# B&R Automation Studio project AxisControl
Automation Studio 4.12.5.95 SP; Templates  para control de eje Maestro y eje esclavo; technology packages: Acp10Arnc0 5.24.1

## Configuration Config1

CPU X20CP1586, AutomationRuntime B4.93, Build 4.1.2, Vc V4.73.1

### Task classes (Cpu.sw)
```
NcDataObjects: acp10etxen <- AxisObjects.acp10etxen.dob, VAxInit <- AxisObjects.Virtual.VAxInit.dob, AcpParTab <- AxisObjects.Real.AcpParTab.dob, AxInit <- AxisObjects.Real.AxInit.dob
Libraries: Acp10man, Acp10par, NcGlobal, Acp10sim, Acp10_MC, sys_lib, brsystem, runtime, MpAxis, MpBase, MpCom
```

### Hardware
```
8BVIxxxxxxDx.xxx-x : 8BVIxxxxxxDx.xxx-x v2.3.0.1  [PLK1 -> X20CP1586.IF3 (NodeNumber=1) [Cable Type=PowerlinkCable, Length=10, Version=1.0.0.3]]
  MotionTP = Acp10Arnc0
  Simulate = standard
X20CP1586 : X20CP1586 v1.10.0.0
  Connector IF2:
    ActivateDevice = 1
  ConfigurationID = AxisControl_Config1
  Simulation = 1
  TimerDeviceType = EPLX2X
  TimerDevice = X20CP1586.IF3
  TaskClassIdleTime = 2000
  FileDevice1
  FileDeviceName1 = USER
  FileDevicePath1 = USER_PATH
```

### Acp10cfg.ncc - X20CP1586/Motion/Acp10cfg.ncc
```
NcConfiguration (Version=5.24.1, NcSwId=Acp10)
  ACP10CF1_typ:
    cnt_nettrc_rec_drive = 1500
    bufsize_trace_upload = 1200
    tc_nc_man_task = Cyclic #1
    glob_pv_as_ncobject = Yes
    ncsys_dl_broadcast = Yes
    ncsys_dl_acp_reset = Yes
    safemc_log_err_to_ax = Yes
    network_init:
      ncsw_init_execute = Yes
      automatic_execute = No
      node_nr_warning = Yes
      net_err_before_ncact = Yes
    nettrc:
      enter_parsecrec = Yes
      enter_ncaction = Yes
      save_ring_startidx = Yes
    cam_prof_download:
      cam_dat_dl_parallel = No
      tc_cam_dl_parallel = Task class for NC Manager task
    plk_if[0]:
      if_name = IF3
      tc_CycDat_PLCopen = Task class for NC Manager task
      mc_broadcast_extdat = No
```

### Acp10map.ncm - X20CP1586/Motion/Acp10map.ncm
```
NcMapping (NcSwId=Acp10, DisabledNodesAreHidden=False)
  NcObject gAxis01 (ModuleId=8BVIxxxxxxDx.xxx-x, Type=ncAXIS, Channel=1, AcoposSimulation=Off, InitParameter=AxInit, AcoposParameter=AcpParTab, Disabled=FALSE, ModuleDisabled=FALSE)
  NcObject gAxis02 (ModuleId=8BVIxxxxxxDx.xxx-x, Type=ncAXIS, Channel=2, AcoposSimulation=Off, InitParameter=AxInit, AcoposParameter=AcpParTab, Disabled=FALSE, ModuleDisabled=FALSE)
  NcObject gVMaster (ModuleId=8BVIxxxxxxDx.xxx-x, Type=ncV_AXIS, Channel=1, InitParameter=VAxInit, Disabled=FALSE, ModuleDisabled=FALSE)
  NcObject gVStep (ModuleId=8BVIxxxxxxDx.xxx-x, Type=ncV_AXIS, Channel=2, InitParameter=VAxInit, Disabled=FALSE, ModuleDisabled=FALSE)
```

### Config.mpaxisbasic - X20CP1586/Motion/Config.mpaxisbasic
```
Element gVMasterLink (Type=mpaxisbasic)
  AxisConfiguration = AxisWithConfiguration
    Drive:
      Controller:
        LoopFilters:
          [0]
          [1]
          [2]
Element gVStepLink (Type=mpaxisbasic)
  AxisConfiguration = AxisWithConfiguration
    Drive:
      Controller:
        LoopFilters:
          [0]
          [1]
          [2]
Element gRealAxisLink_1 (Type=mpaxisbasic)
  AxisConfiguration = AxisWithConfiguration
    Drive:
      Controller:
        LoopFilters:
          [0]
          [1]
          [2]
Element gRealAxisLink_2 (Type=mpaxisbasic)
  AxisConfiguration = AxisWithConfiguration
    Drive:
      Controller:
        LoopFilters:
          [0]
          [1]
          [2]
```

## Logical view

Binary libraries used (declarations not repeated): operator, runtime, astime, AsIecCon, Acp10man, Acp10par, NcGlobal, Acp10sim, Acp10_MC, sys_lib, brsystem, MpAxis, MpBase, MpCom, standard

### Global.typ - Global data types
```iecst
TYPE
	Axis_type : 	STRUCT
		Enable : BOOL; (*Habilita Control Global del eje*)
		Cmd : AxisComand_type;
		Sts : AxisStatus_type;
		Par : AxisParameters_type;
	END_STRUCT;
	AxisComand_type : 	STRUCT
		Enable : BOOL;
		Reset : BOOL;
		ConfigReq : BOOL;
	END_STRUCT;
	AxisStatus_type : 	STRUCT
		ConfigDone : BOOL;
		Error : BOOL;
	END_STRUCT;
	AxisParameters_type : 	STRUCT
		New_Member : USINT;
	END_STRUCT;
END_TYPE
```

### Global.var - Global variables
```iecst
(*Declariacion Ejes *)
VAR
	gAxis01 : ACP10AXIS_typ;
	gAxis02 : ACP10AXIS_typ;
	gVMaster : ACP10VAXIS_typ;
	gVStep : ACP10VAXIS_typ;
END_VAR
(*UDT Control dej Eje*)
VAR
	gAxis : ARRAY[0..MAX_AXIS] OF Axis_type;
END_VAR
```

### Constant.var - Global Constant
```iecst
(*Asignacion ejes*)
VAR CONSTANT
	VMASTER : USINT := 0;
END_VAR
(*Constantes de control de programa*)
VAR CONSTANT
	MAX_AXIS : USINT := 4; (*Cantidad maxima de ejes *)
END_VAR
```


### Program Logical/VirtualMaster (IEC)

#### Cyclic.st - Cyclic code
```iecst
(*********************************************************************************
 * Copyright:
 * Author:    NoVi
 * Created:   March 28, 2024/4:33 PM
 *********************************************************************************)

PROGRAM _CYCLIC

	//------ Subrutinas ------//

	Config;

	///////////////////////////

	//----- Habilita el Eje ------//

	AxisBasic.Enable 	:= gAxis[AxisIndex].Enable;
	AxisConfig.Enable 	:= AxisBasic.Active;
	AxisCam.Enable 		:= AxisBasic.Active AND AxisIndex > VMASTER;

	////////////////////////////////

	CASE StAxis OF

		STATE_INIT:

			IF AxisBasic.Active AND AxisBasic.Info.BootState = mpAXIS_BLP_DONE AND AxisBasic.Info.ReadyToPowerOn AND AxisConfig.Active THEN
				StAxis := STATE_CONFIG;
			END_IF

		STATE_ERROR:

	END_CASE

	//----- Administracion de Errores ------//

	gAxis[AxisIndex].Sts.Error := AxisBasic.Error OR AxisConfig.Error OR AxisCam.Error;

	IF gAxis[AxisIndex].Sts.Error THEN
		StAxis := STATE_ERROR;
	END_IF

	//-- Reset
	AxisBasic.ErrorReset 	:= AxisBasic.Error AND gAxis[AxisIndex].Cmd.Reset;
	AxisConfig.ErrorReset 	:= AxisConfig.Error AND gAxis[AxisIndex].Cmd.Reset;
	AxisCam.ErrorReset		:= AxisCam.Error AND gAxis[AxisIndex].Cmd.Reset;

	///////////////////////////////////////////

END_PROGRAM
```

#### Config.st
```iecst
(*********************************************************************************
 * Copyright:
 * Author:    aleja
 * Created:   March 29, 2024/1:46 PM
 *********************************************************************************)

ACTION Config:

	//---- Numero del Eje ----///
	AxisIndex := VMASTER;

	//---- Nombre del eje ----//
	AxisName := 'Virtual Master';

	//---- Hablita el eje ----//
	gAxis[AxisIndex].Enable := TRUE; // ESTE DATA DEBERA SER USADO EN UN VARIABLE DE LA CONFIGURACION MAQUINA PARA HABILITAR O DESHABILITAR UN EJE.

	//---- Limite de velocidad -----//
	LimitSpeed 	:= 6600.0;

	//----- Limete de aceleracion/desaceleracion ----//
	LimitAccDec := 6600.0;

	//---- Relacion de velocoidad motor/reductor ----//
	GearIn 	:= 1;
	GearOut := 1;

	//---- Seleccion direccion de rotacion del eje ----//
	AxisDirection := TRUE; // TRUE = sentido de las manesillas del reloj; FALSE = en contra de las manesillas del reloj;

	// ---- Definicion sentido de giro del eje ----//
	IF AxisDirection THEN
		Direction	:= mpAXIS_DIR_CLOCKWISE;
	ELSE
		Direction	:= mpAXIS_DIR_COUNTERCLOCKWISE;
	END_IF

	// ---- Definicion Paramentros de posicion del eje ----//
	Period :=  360.0;
	SectorNumber := 1;
	ReferenceDistance := Period * SectorNumber;

	IF gAxis[AxisIndex].Cmd.ConfigReq THEN

		AxisConfigPar.AxisName := AxisName ;

		//Axis
		AxisConfigPar.Axis.BaseType 				:= mpAXIS_PERIODIC_ROTARY;
		AxisConfigPar.Axis.MeasurementUnit 			:= mpAXIS_UNIT_GENERIC;
		AxisConfigPar.Axis.MeasurementResolution 	:= 0.01;
		AxisConfigPar.Axis.PeriodSettings.Period	:= Period; // Valor con fines de prueba este deberia estar en 360 ya que es el VMaster

		AxisConfigPar.Axis.MovementLimits.VelocityPositive	:= LimitSpeed;
		AxisConfigPar.Axis.MovementLimits.VelocityNegative	:= LimitSpeed;
		AxisConfigPar.Axis.MovementLimits.Acceleration		:= LimitAccDec;
		AxisConfigPar.Axis.MovementLimits.Deceleration		:= LimitAccDec;

		//Drive
		AxisConfigPar.Drive.Gearbox.Input			:= GearIn;
		AxisConfigPar.Drive.Gearbox.Output			:= GearOut;
		AxisConfigPar.Drive.Gearbox.Direction 		:= Direction;
		AxisConfigPar.Drive.Transformation.ReferenceDistance := ReferenceDistance;

		gAxis[AxisIndex].Sts.ConfigDone := TRUE;

	END_IF

	////---- Limites asignados jog ----////

	gAxis[AxisIndex].Par.Jog.Acc 	:= LIMIT(MIN_ACC_DECEL_JOG,gAxis[AxisIndex].Par.Jog.Acc,MAX_ACC_DECEL_JOG);
	gAxis[AxisIndex].Par.Jog.Decel 	:= LIMIT(MIN_ACC_DECEL_JOG,gAxis[AxisIndex].Par.Jog.Decel,MAX_ACC_DECEL_JOG);
	gAxis[AxisIndex].Par.Jog.Speed 	:= LIMIT(MIN_SPEED_JOG,gAxis[AxisIndex].Par.Jog.Speed,MAX_SPEED_JOG);

	////---- FB Control del eje -----////

	AxisBasic.Axis 				:= ADR(gVMaster);
	AxisBasic.MpLink 			:= ADR(gVMasterLink);
	AxisBasic.Parameters 		:= ADR(AxisBasicPar);
	AxisBasic();

	AxisConfig.MpLink 			:= ADR(gVMasterLink);
	AxisConfig.Configuration 	:= ADR(AxisConfigPar);
	AxisConfig();

	AxisCam.MpLink				:= ADR(gVMasterLink);
	AxisCam.MpLinkMaster		:= 0;
	AxisCam.Parameters			:= ADR(AxisCamPar);
	AxisCam();

END_ACTION
```

#### Types.typ - Local data types
```iecst
TYPE
	AxisStates_enum :
		(
		STATE_INIT := 0, (*INICIO DE SECUENCIA DEL EJE*)
		STATE_CONFIG := 10, (*CONFIGURACION DEL EJE*)
		STATE_ERROR := 9000 (*EJE EN ERROR*)
		);
END_TYPE
```

#### Variables.var - Local variables
```iecst
(*Motion FBs*)
VAR
	AxisBasic : MpAxisBasic;
	AxisBasicPar : MpAxisBasicParType;
	AxisConfig : MpAxisBasicConfig;
	AxisConfigPar : MpAxisBasicConfigType;
	AxisCam : MpAxisCamSequencer;
	AxisCamPar : MpAxisCamSequencerParType;
END_VAR
(*Variables de control *)
VAR
	Direction : MpAxisMotorDirectionEnum;
	AxisConfigDone : BOOL;
	AxisConfigReq : BOOL;
	LimitSpeed : REAL;
	LimitAccDec : REAL;
	GearIn : UDINT;
	GearOut : UDINT;
	AxisDirection : BOOL;
	AxisName : STRING[20];
	Period : LREAL;
	ReferenceDistance : LREAL;
	SectorNumber : LREAL;
	AxisIndex : USINT;
	AccVal : REAL;
	DecelVal : REAL;
END_VAR
(*Variables control de secuancias*)
VAR
	StAxis : AxisStates_enum; (*Esatdos del control del Eje*)
	StConfig : ConfigStates_enum;
	StHome : HomeState_enum;
	StMoveAbsolute : AbsoluteMov_enum;
	StJog : JogStates_enum;
	StMoveAdditive : AdditiveMov_enum;
	StMoveVelocity : VelocityMov_enum;
END_VAR
(*Variables secuencia JOG*)
VAR
	TON_Jog : TON;
	AuxJogStop : BOOL;
	R_Reset : R_TRIG;
END_VAR
```

#### Constants.var - Local Constants
```iecst
(*INDICES*)
VAR CONSTANT
	MASTER : USINT := 0; (*NUMERO DE INDICE ASIGNADO AL EJE MAESTRO *)
END_VAR
(*CONSTANTES JOG*)
VAR CONSTANT
	JOG_TIME : TIME := T#4S;
	MAX_ACC_DECEL_JOG : REAL := 1000.0;
	MIN_ACC_DECEL_JOG : REAL := 100.0;
	MIN_SPEED_JOG : REAL := 10.0;
	MAX_SPEED_JOG : REAL := 400.0;
END_VAR
```

### AxisControl_VirtualMaster.txt
```
CONTROL DE EJE MAESTRO
Estados de la secuencia de control

0 .- Habilitar el Eje [STATE_INIT]:

el eje debe ser habilitado en la "Action" Config.st, por medio de la variable gAxis[AxisIndex].Enable

9000 .- Control de Error [STATE_ERROR]; para que que se de un error es necesario que un bloque de funcion de control tenga la salida error = TRUE;
		para restablecer el error la variable gAxis[AxisIndex].Cmd.Reset = TRUE,
```

Listed in the project but not available here: Logical/VirtualMaster/Init.st, Logical/VirtualMaster/Exit.st, Logical/AxisObjects/Virtual, Logical/AxisObjects/Real, Logical/AxisObjects/acp10etxen
